TYPE ST_WriterInternalState :
STRUCT
    nBufferSize         : UDINT;                // Size of the current buffer
    nBufferPos          : UDINT;                // The position within the current buffer (i.e. the next byte to read)
    bError              : BOOL;
    pCodedOutputStream  : POINTER TO FB_CodedOutputStream;
    eWriterErrorCode    : E_WriterErrorCode;    // 0 = no error, <> 0 = error
END_STRUCT
END_TYPE

(* stored: Version 1.1.0.1
   DUT ST_WriterInternalState: Id {f65f559f-4118-4f64-8be6-cf1721b70ddd} *)
